// TIA Portal V20 export
VAR_GLOBAL   // PLC tag table "LKinCtrl_HMI_Shared_Interlocks"
END_VAR
VAR_GLOBAL CONSTANT   // user constants
   LKINCTRL_INTERLOCKID_EXTERNALINTERLOCK : Int := 8000;
   LKINCTRL_INTERLOCKID_NONE : Int := 0;
   LKINCTRL_INTERLOCKID_OPERATIONMODE : Int := 8001;
END_VAR
